TYPE E_RobotStateTM :
(
	READY,
	PREPARATION,
	SEND
) UDINT;
END_TYPE

(* stored: Version 1.1.0.1, ProductVersion 3.1.4024.11
   DUT E_RobotStateTM: Id {18e32e38-b246-4929-b93a-0d75c5d81c23} *)
